(* PLC project ForceTraceReferenceTypes, BPP Internal Engineering BPP reference types 0.2.0.0 *)
(* stored: creationDateTime 2026-09-15T00:00:00, modificationDateTime 2026-09-15T00:00:00 *)

TYPE ForceTraceReferenceSettings : STRUCT
  ThresholdN : REAL := 2500;
  LimitN : REAL := 0;
  WindowMs : DINT := 1000;
  TimeoutMs : DINT := 30000;
END_STRUCT;
END_TYPE

TYPE ForceTraceReferenceSignals : STRUCT
  ForceN : REAL := 0;
  QualityGood : BOOL := false;
  Measuring : BOOL := false;
END_STRUCT;
END_TYPE
